# EPICS substitutions: zoomBuilder/iocs/BL99I-LCH-IOC-01/BL99I-LCH-IOC-01App/Db/BL99I-LCH-IOC-01_expanded.substitutions
# This file was automatically generated on Mon 15 Oct 2018 09:44:11 BST from
# source: /home/jjc62351/work/Zoom/zoomBuilder/etc/makeIocs/BL99I-LCH-IOC-01.xml
#
# *** Please do not edit this file: edit the source file instead. ***
#

# Macros:
#  PORT      The asyn port for the pmac controller
#  P         PV Prefix
#  NAXES     Number of axes
#  TIMEOUT   Timeout for controller communication
#  FEEDRATE  feedrate below which we go into error
#  CSG0      Name for Coordinate System Group 0
#  CSG1      Name for Coordinate System Group 1
#  CSG2      Name for Coordinate System Group 2
#  CSG3      Name for Coordinate System Group 3
#  CSG4      Name for Coordinate System Group 4
#  CSG5      Name for Coordinate System Group 5
#  CSG6      Name for Coordinate System Group 6
#  CSG7      Name for Coordinate System Group 7
file $(PMAC)/db/pmacController.template
{
pattern { PORT, P, NAXES, TIMEOUT, FEEDRATE, CSG0, CSG1, CSG2, CSG3, CSG4, CSG5, CSG6, CSG7 }
    { "BRICK1", "BL99I-LCH-STEP-01", "8", "4", "100", "", "", "", "", "", "", "", "" }
}

# Macros:
#  PORT  The asyn port for the pmac controller
#  P     PV Prefix
file $(PMAC)/db/pmacStatus.template
{
pattern { PORT, P }
    { "BRICK1", "BL99I-LCH-STEP-01" }
}

# Macros:
#  PMAC  Pmac/Geobrick name
#  AXIS  Axis number
#  PORT  Asyn port
file $(PMAC)/db/pmacStatusAxis.template
{
pattern { PMAC, AXIS, PORT }
    { "BL99I-LCH-STEP-01", "1", "BRICK1" }
    { "BL99I-LCH-STEP-01", "2", "BRICK1" }
    { "BL99I-LCH-STEP-01", "3", "BRICK1" }
    { "BL99I-LCH-STEP-01", "4", "BRICK1" }
    { "BL99I-LCH-STEP-01", "5", "BRICK1" }
    { "BL99I-LCH-STEP-01", "6", "BRICK1" }
    { "BL99I-LCH-STEP-01", "7", "BRICK1" }
    { "BL99I-LCH-STEP-01", "8", "BRICK1" }
}

# Macros:
#  P                Device Prefix
#  M                Device Suffix
#  PORT             Delta tau motor controller
#  ADDR             Address on controller
#  DESC             Description, displayed on EDM screen
#  MRES             Motor Step Size (EGU)
#  VELO             Velocity (EGU/s)
#  PREC             Display Precision
#  EGU              Engineering Units
#  TWV              Tweak Step Size (EGU)
#  DTYP             DTYP of record
#  DIR              User Direction
#  VBAS             Base Velocity (EGU/s)
#  VMAX             Max Velocity (EGU/s), defaults to VELO
#  ACCL             Seconds to Velocity
#  BDST             BL Distance (EGU)
#  BVEL             BL Velocity (EGU/s)
#  BACC             BL Seconds to Veloc.
#  DHLM             Dial High Limit
#  DLLM             Dial Low Limit
#  HLM              User High Limit
#  LLM              User Low Limit
#  HLSV             HW Lim. Violation Svr
#  INIT             Startup commands
#  SREV             Steps per Revolution
#  RRES             Readback Step Size (EGU)
#  ERES             Encoder Step Size (EGU)
#  JAR              Jog Acceleration (EGU/s^2)
#  UEIP             Use Encoder If Present
#  URIP             Use RDBL If Present
#  RDBL             Readback Location, set URIP = 1 if you specify this
#  RLNK             Readback output link
#  RTRY             Max retry count
#  DLY              Readback settle time (s)
#  OFF              User Offset (EGU)
#  RDBD             Retry Deadband (EGU)
#  FOFF             Freeze Offset, 0=variable, 1=frozen
#  ADEL             Alarm monitor deadband (EGU)
#  NTM              New Target Monitor, only set to 0 for soft motors
#  FEHIGH           HIGH limit for following error
#  FEHIHI           HIHI limit for following error
#  FEHHSV           HIHI alarm severity for following error
#  FEHSV            HIGH alarm severity for following error
#  SCALE            Scale factor, if pmacSetAxisScale is used this should be set
#  HOMEVIS          If 1 then home is visible on the gui
#  HOMEVISSTR       If HOMEVIS=0, then display this text on the gui instead
#  name             Object name and gui association name
#  alh              Set this to alh to add the motor to the alarm handler and send emails,
#  gda_name         Name to export this as to GDA
#  gda_desc         Description to export this as to GDA
#  SPORT            Delta tau motor controller comms port
#  HOME             Prefix for autohome instance. Defaults to $(P). If unspecified,
#  ALLOW_HOMED_SET  Set to a blank to allow this axis to have its homed
file $(PMAC)/db/dls_pmac_asyn_motor.template
{
pattern { P, M, PORT, ADDR, DESC, MRES, VELO, PREC, EGU, TWV, DTYP, DIR, VBAS, VMAX, ACCL, BDST, BVEL, BACC, DHLM, DLLM, HLM, LLM, HLSV, INIT, SREV, RRES, ERES, JAR, UEIP, URIP, RDBL, RLNK, RTRY, DLY, OFF, RDBD, FOFF, ADEL, NTM, FEHIGH, FEHIHI, FEHHSV, FEHSV, SCALE, HOMEVIS, HOMEVISSTR, name, alh, gda_name, gda_desc, SPORT, HOME, PMAC, ALLOW_HOMED_SET }
    { "BL99I-LCH-MO-01", ":ZOOM:LENS1", "BRICK1", "1", "Zoom lens 1", "0.0004", "2", "3", "mm", "0.1", "asynMotor", "0", "0", "$(VELO)", "0.5", "0", "0", "", "20.468", "-15.892", "36.4", "0.04", "MAJOR", "", "1000", "", "", "", "0", "0", "", "", "0", "0", "15.9316", "", "0", "0", "1", "0", "0", "NO_ALARM", "NO_ALARM", "1", "1", "Use motor summary screen", "ZOOML1", "None", "", "$(DESC)", "BRICK1port", "$(P)", "BL99I-LCH-STEP-01", "#" }
    { "BL99I-LCH-MO-01", ":ZOOM:LENS2", "BRICK1", "2", "Zoom lens 2", "0.0004", "2", "3", "mm", "0.1", "asynMotor", "0", "0", "$(VELO)", "0.5", "0", "0", "", "14.468", "-24.732", "56.4", "17.2", "MAJOR", "", "1000", "", "", "", "0", "0", "", "", "0", "0", "41.9316", "", "0", "0", "1", "0", "0", "NO_ALARM", "NO_ALARM", "1", "1", "Use motor summary screen", "ZOOML2", "None", "", "$(DESC)", "BRICK1port", "$(P)", "BL99I-LCH-STEP-01", "#" }
}

# Macros:
#  PORT     The asyn port for the pmac cs controller
#  PMAC     PV Prefix for the motor controller
#  CS       Coordinate System Number for the cs controller
#  TIMEOUT  Timeout for controller communication
file $(PMAC)/db/pmacCsController.template
{
pattern { PORT, PMAC, CS, TIMEOUT }
    { "CS3", "BL99I-LCH-STEP-01", "3", "4" }
}

# Macros:
#  P           Device Prefix
#  M           Device Suffix
#  PORT        Delta tau motor controller
#  ADDR        Address on controller
#  DESC        Description, displayed on EDM screen
#  MRES        Motor Step Size (EGU)
#  VELO        Velocity (EGU/s)
#  PREC        Display Precision
#  EGU         Engineering Units
#  TWV         Tweak Step Size (EGU)
#  DTYP        DTYP of record
#  DIR         User Direction
#  VBAS        Base Velocity (EGU/s)
#  VMAX        Max Velocity (EGU/s), defaults to VELO
#  ACCL        Seconds to Velocity
#  BDST        BL Distance (EGU)
#  BVEL        BL Velocity (EGU/s)
#  BACC        BL Seconds to Veloc.
#  DHLM        Dial High Limit
#  DLLM        Dial Low Limit
#  HLM         User High Limit
#  LLM         User Low Limit
#  HLSV        HW Lim. Violation Svr
#  INIT        Startup commands
#  SREV        Steps per Revolution
#  RRES        Readback Step Size (EGU)
#  ERES        Encoder Step Size (EGU)
#  JAR         Jog Acceleration (EGU/s^2)
#  UEIP        Use Encoder If Present
#  URIP        Use RDBL If Present
#  RDBL        Readback Location, set URIP = 1 if you specify this
#  RLNK        Readback output link
#  RTRY        Max retry count
#  DLY         Readback settle time (s)
#  OFF         User Offset (EGU)
#  RDBD        Retry Deadband (EGU)
#  FOFF        Freeze Offset, 0=variable, 1=frozen
#  ADEL        Alarm monitor deadband (EGU)
#  NTM         New Target Monitor, only set to 0 for soft motors
#  FEHIGH      HIGH limit for following error
#  FEHIHI      HIHI limit for following error
#  FEHHSV      HIHI alarm severity for following error
#  FEHSV       HIGH alarm severity for following error
#  SCALE       Scale factor, if pmacSetAxisScale is used this should be set
#  HOMEVIS     If 1 then home is visible on the gui
#  HOMEVISSTR  If HOMEVIS=0, then display this text on the gui instead
#  name        Object name and gui association name
#  alh         Set this to alh to add the motor to the alarm handler and send emails,
#  gda_name    Name to export this as to GDA
#  gda_desc    Description to export this as to GDA
file $(PMAC)/db/dls_pmac_cs_asyn_motor.template
{
pattern { P, M, PORT, ADDR, DESC, MRES, VELO, PREC, EGU, TWV, DTYP, DIR, VBAS, VMAX, ACCL, BDST, BVEL, BACC, DHLM, DLLM, HLM, LLM, HLSV, INIT, SREV, RRES, ERES, JAR, UEIP, URIP, RDBL, RLNK, RTRY, DLY, OFF, RDBD, FOFF, ADEL, NTM, FEHIGH, FEHIHI, FEHHSV, FEHSV, SCALE, HOMEVIS, HOMEVISSTR, name, alh, gda_name, gda_desc, PMAC, CS }
    { "BL99I-LCH-MO-01", ":ZOOM:GAP", "CS3", "8", "Zoom gap", "0.0001", "1", "3", "mm", "1", "asynMotor", "0", "0", "$(VELO)", "0.5", "0", "0", "", "17", "2", "17", "2", "MAJOR", "", "1000", "", "", "", "0", "0", "", "", "0", "0", "0", "", "0", "0", "1", "0", "0", "NO_ALARM", "NO_ALARM", "1", "1", "Use motor summary screen", "", "None", "", "$(DESC)", "BL99I-LCH-STEP-01", "3" }
    { "BL99I-LCH-MO-01", ":ZOOM:CENTRE", "CS3", "7", "Zoom cen", "0.0001", "1", "3", "mm", "1", "asynMotor", "0", "0", "$(VELO)", "0.5", "0", "0", "", "42.5", "13", "42.5", "13", "MAJOR", "", "1000", "", "", "", "0", "0", "", "", "0", "0", "0", "", "0", "0", "1", "0", "0", "NO_ALARM", "NO_ALARM", "1", "1", "Use motor summary screen", "", "None", "", "$(DESC)", "BL99I-LCH-STEP-01", "3" }
}
